// TIA Portal V20 export
VAR_GLOBAL   // PLC tag table "EVT_Const_Gen"
END_VAR
VAR_GLOBAL CONSTANT   // user constants
   EVT_CAPACITY : Int := 1000;   // EVTLOG entries / EVTLOG 항목 수
   EVT_LAST : Int := 999;   // EVTLOG.Entry upper bound / EVTLOG.Entry 상한
   EVT_MIN_LEVEL_DEFAULT : USInt := 2;   // Default Cfg.MinLevel / Cfg.MinLevel 기본값
   EVT_MAX_PER_SCAN_DEFAULT : Int := 32;   // Default Cfg.MaxPerScan / Cfg.MaxPerScan 기본값
   EVT_CATMASK_ALL : DWord := 16#0003FFFE;   // Cfg.CatMask, every category / Cfg.CatMask 전 분류
   EVT_LVL_TRACE : USInt := 0;   // Level TRACE / 레벨 TRACE
   EVT_LVL_DEBUG : USInt := 1;   // Level DEBUG / 레벨 DEBUG
   EVT_LVL_INFO : USInt := 2;   // Level INFO / 레벨 INFO
   EVT_LVL_WARN : USInt := 3;   // Level WARN / 레벨 WARN
   EVT_LVL_ERROR : USInt := 4;   // Level ERROR / 레벨 ERROR
   EVT_CAT_SYS : USInt := 1;   // Category SYS (CatMask bit 1) / 분류 SYS
   EVT_CAT_MODE : USInt := 2;   // Category MODE (CatMask bit 2) / 분류 MODE
   EVT_CAT_STEP : USInt := 3;   // Category STEP (CatMask bit 3) / 분류 STEP
   EVT_CAT_TASK : USInt := 4;   // Category TASK (CatMask bit 4) / 분류 TASK
   EVT_CAT_CMD : USInt := 5;   // Category CMD (CatMask bit 5) / 분류 CMD
   EVT_CAT_ALARM : USInt := 6;   // Category ALARM (CatMask bit 6) / 분류 ALARM
   EVT_CAT_GRIP : USInt := 7;   // Category GRIP (CatMask bit 7) / 분류 GRIP
   EVT_CAT_DRIVE : USInt := 8;   // Category DRIVE (CatMask bit 8) / 분류 DRIVE
   EVT_CAT_SAFETY : USInt := 9;   // Category SAFETY (CatMask bit 9) / 분류 SAFETY
   EVT_CAT_SENSOR : USInt := 10;   // Category SENSOR (CatMask bit 10) / 분류 SENSOR
   EVT_CAT_MEAS : USInt := 11;   // Category MEAS (CatMask bit 11) / 분류 MEAS
   EVT_CAT_ILOCK : USInt := 12;   // Category ILOCK (CatMask bit 12) / 분류 ILOCK
   EVT_CAT_ANTICOL : USInt := 13;   // Category ANTICOL (CatMask bit 13) / 분류 ANTICOL
   EVT_CAT_COMM : USInt := 14;   // Category COMM (CatMask bit 14) / 분류 COMM
   EVT_CAT_DATA : USInt := 15;   // Category DATA (CatMask bit 15) / 분류 DATA
   EVT_CAT_STATION : USInt := 16;   // Category STATION (CatMask bit 16) / 분류 STATION
   EVT_CAT_SCEN : USInt := 17;   // Category SCEN (CatMask bit 17) / 분류 SCEN
   EVT_SYS_STARTUP : UInt := 101;   // SYS INFO / PLC 기동 {a:bits:startup}
   EVT_SYS_PROG_ERROR : UInt := 102;   // SYS ERROR / Programming error : block {src}, Fault_ID {a:hex}, DB {b}
   EVT_SYS_CYCLE_OVERRUN : UInt := 103;   // SYS ERROR / Cycle time error : Fault_ID {a:hex}
   EVT_SYS_CLOCK_SET : UInt := 104;   // SYS WARN / 시계 보정 {a} ms
   EVT_SYS_LOGGER_DROP : UInt := 105;   // SYS WARN / 로거 누락 : Dropped {a} (MaxPerScan 초과)
   EVT_SYS_LOGGER_SLOW : UInt := 106;   // SYS WARN / 로거 실행 시간 MaxRunUs {a} µs
   EVT_MODE_CHANGED : UInt := 201;   // MODE INFO / {b:mode} → {a:mode}
   EVT_MODE_REJECTED : UInt := 202;   // MODE WARN / 모드 요청 거부 {b:mode} → {a:mode}
   EVT_MODE_AUTO_STOP : UInt := 203;   // MODE INFO / AUTO 정지 : {a:auto_stop}
   EVT_MODE_AUTO_START : UInt := 204;   // MODE INFO / AUTO 시작 : {a:start_src}
   EVT_MODE_AUTO_REFUSED : UInt := 205;   // MODE WARN / AUTO 시작 불가 : {a:bits:start_block}
   EVT_MODE_FAULT_RESET : UInt := 206;   // MODE INFO / Fault reset {a:reset_result} (FaultCode[0] {b})
   EVT_MODE_OPTION : UInt := 207;   // MODE WARN / Option {src:option} {a:onoff}
   EVT_MODE_TEACH_BUFF_CLEARED : UInt := 208;   // MODE WARN / Teach 진입 : TASK.Buff {a} 건 삭제
   EVT_MODE_GCS_ONLINE : UInt := 209;   // MODE INFO / GCS_Online {a:onoff}
   EVT_MODE_GRM_PANEL : UInt := 210;   // MODE INFO / GRM {src:grm_panel} {a:onoff}
   EVT_MODE_STATUS_BIT : UInt := 211;   // MODE DEBUG / Status.{src:machine_status} {a:onoff}
   EVT_TASK_ACCEPTED : UInt := 401;   // TASK INFO / 수락 {src:task_type} · Cell {a} · WorkId {b}
   EVT_TASK_REJECTED : UInt := 402;   // TASK WARN / 거부 {src:task_type} : {a:bits:reject} ({b:validation})
   EVT_TASK_HEADER_TIMEOUT : UInt := 403;   // TASK ERROR / 명령 헤더 빈 필드 15 s (F{a})
   EVT_TASK_LOADED : UInt := 404;   // TASK INFO / 시작 {src:task_type} · Cell {a} · WorkId {b}
   EVT_TASK_WAIT_DEADLOCK : UInt := 405;   // TASK WARN / 적재 대기 : 상대 로봇 교착·회피 {a} ms
   EVT_TASK_RESUMED : UInt := 406;   // TASK INFO / 정지 후 재개 → step {a}
   EVT_TASK_CROSSCHECK_FAIL : UInt := 407;   // TASK ERROR / 아이템 교차 확인 실패 F{a}
   EVT_TASK_COMPLETED : UInt := 408;   // TASK INFO / 완료 {src:task_type} · Cell {a} · WorkId {b}
   EVT_TASK_MANUAL_COMPLETE : UInt := 409;   // TASK INFO / 수동 완료 ({src:cmd_src}) : {a:manual_complete} · WorkId {b}
   EVT_TASK_PENDING_END : UInt := 410;   // TASK INFO / CompletePending 해소 : {a:pending_end} · WorkId {b}
   EVT_TASK_CANCELED : UInt := 411;   // TASK INFO / 취소 ({src:cmd_src}) : {a:cancel_result} · WorkId {b}
   EVT_TASK_CANCEL_IGNORED : UInt := 412;   // TASK WARN / AUTO 중 OPC 취소 무시 · WorkId {b}
   EVT_TASK_RESTART_LAST : UInt := 413;   // TASK INFO / 마지막 작업 재시작 · WorkId {b}
   EVT_TASK_TEACH_OVERRIDE : UInt := 414;   // TASK WARN / TeachOverride : {src:override_kind} {a} 위치 갱신
   EVT_TASK_ITEM_CHANGED : UInt := 415;   // TASK INFO / 잡은 아이템 {b} → {a}
   EVT_TASK_CYCLE : UInt := 416;   // TASK INFO / 사이클 ProcessTime {a} ms · Travel {b} mm (flags {src:hex})
   EVT_TASK_STEP_TIMEOUT : UInt := 417;   // TASK WARN / Step {src:task_step} 타임아웃 : WaitCause {a} ({b} ms)
   EVT_TASK_STATUS_BIT : UInt := 418;   // TASK DEBUG / TASK.Status bit {src} {a:onoff}
   EVT_CMD_ALLSTOP : UInt := 501;   // CMD WARN / AllStop {b:onoff} : {a:bits:stop_src}
   EVT_CMD_EMS : UInt := 502;   // CMD ERROR / AllStop_Fast (EMS) {a:onoff}
   EVT_CMD_RESET : UInt := 503;   // CMD INFO / Reset : {a:bits:stop_src}
   EVT_CMD_GCS_START : UInt := 504;   // CMD INFO / GCS Common.Start
   EVT_CMD_BUZZER_STOP : UInt := 505;   // CMD INFO / BuzzerStop
   EVT_CMD_GRIP_LEARN : UInt := 506;   // CMD INFO / Gripper LearnCmd
   EVT_CMD_UNUSED : UInt := 507;   // CMD WARN / 받았지만 처리하지 않는 명령 : {src:unused_cmd}
   EVT_CMD_RESPONSE : UInt := 508;   // CMD INFO / 응답 {b:task_type} SEQ {a}
   EVT_CMD_HMI_TASK_BUTTON : UInt := 509;   // CMD INFO / HMI {src:hmi_task_button}
   EVT_CMD_FUNCTION : UInt := 510;   // CMD INFO / Function {src:function} {a:onoff}
   EVT_CMD_DRIVE_POWER : UInt := 511;   // CMD INFO / {src:axis} PowerOn {a:onoff} (manual)
   EVT_CMD_MANUAL_START : UInt := 512;   // CMD INFO / Manual {src:manual_start} 시작
   EVT_CMD_JOG : UInt := 513;   // CMD DEBUG / {src:axis} Jog {a:hex}
   EVT_ALM_RAISED : UInt := 601;   // ALARM ERROR / {alarm} 발생 (step {b})
   EVT_ALM_CLEARED : UInt := 602;   // ALARM INFO / {alarm} 해제
   EVT_ALM_RESET : UInt := 603;   // ALARM INFO / {src:alarm_area} reset ({a} bits set)
   EVT_ALM_TO_FAULT : UInt := 604;   // ALARM ERROR / FAULT 전환 : 첫 코드 {a}
   EVT_GRIP_REQ : UInt := 701;   // GRIP INFO / 요청 {src:grip_mode} Target {a/10} mm ({b:grip_owner})
   EVT_GRIP_REJECT : UInt := 702;   // GRIP WARN / 요청 거부 {a:grip_err} ({src:grip_owner})
   EVT_GRIP_ABORT : UInt := 703;   // GRIP WARN / 요청 중단 ({src:grip_owner})
   EVT_GRIP_ERROR : UInt := 704;   // GRIP WARN / 실패 {src:grip_err} StopPos {a/10} mm · {b} %
   EVT_GRIP_STATUS : UInt := 705;   // GRIP WARN / {src:grip_status} {a}
   EVT_GRIP_RETRY : UInt := 706;   // GRIP INFO / 재파지 {a} → step {b}
   EVT_GRIP_LEARN : UInt := 707;   // GRIP INFO / Learn {src:learn_phase} LearnError {a} @ {b/10} mm
   EVT_GRIP_THERMAL : UInt := 708;   // GRIP WARN / Thermal {a:onoff}
   EVT_GRIP_STATE : UInt := 709;   // GRIP DEBUG / {b:grip_state} → {a:grip_state}
   EVT_GRIP_ITEM_DETECT : UInt := 710;   // GRIP DEBUG / ItemDetect {a:onoff}
   EVT_GRIP_STEP : UInt := 711;   // GRIP DEBUG / GRIP.Step {b} → {a}
   EVT_GRIP_READY : UInt := 712;   // GRIP WARN / Sense.Ready {a:onoff}
   EVT_DRV_FAULT : UInt := 801;   // DRIVE ERROR / {src:axis} Fault MainCode {a} SubCode {b}
   EVT_DRV_WARNING : UInt := 802;   // DRIVE WARN / {src:axis} Warning MainCode {a} SubCode {b}
   EVT_DRV_FAULT_CLEARED : UInt := 803;   // DRIVE INFO / {src:axis} Fault/Warning 해제
   EVT_DRV_REF_LOST : UInt := 804;   // DRIVE ERROR / {src:axis} Referenced 상실
   EVT_DRV_OVERHEAT : UInt := 805;   // DRIVE WARN / {src:axis} Overheat {a:bits:overheat}
   EVT_DRV_SYNC : UInt := 806;   // DRIVE WARN / X1/X2 sync F{a} (SyncDiff {b/10} mm)
   EVT_DRV_LAG : UInt := 807;   // DRIVE WARN / X lag {a/10} mm ({b:alarm_area})
   EVT_DRV_ENABLE_FAIL : UInt := 808;   // DRIVE ERROR / {src:axis} Enable / encoder F{a}
   EVT_DRV_LIMIT : UInt := 809;   // DRIVE WARN / {src:axis} limit {a:bits:limit}
   EVT_DRV_MDR : UInt := 810;   // DRIVE WARN / MDR {a:bits:mdr}
   EVT_DRV_STATE : UInt := 811;   // DRIVE DEBUG / {src:axis} {a:bits:drive_state}
   EVT_DRV_HOMING_DONE : UInt := 812;   // DRIVE INFO / {src:axis} homing 완료
   EVT_DRV_TARGET_RANGE : UInt := 813;   // DRIVE ERROR / {src:axis} 목표 범위 밖 F{a} (target {b/10} mm)
   EVT_SAFE_EMS : UInt := 901;   // SAFETY ERROR / EMS {a:onoff}
   EVT_SAFE_INPUT : UInt := 902;   // SAFETY WARN / {src:safety_input} {a:onoff}
   EVT_SAFE_IO_FORCE : UInt := 903;   // SAFETY WARN / {src:io_force} {a:onoff}
   EVT_SAFE_OUTPUT : UInt := 904;   // SAFETY DEBUG / Output {src:output} {a:onoff}
   EVT_SNS_MODULE : UInt := 1001;   // SENSOR WARN / Module {src:module} {a:onoff}
   EVT_SNS_BELT : UInt := 1002;   // SENSOR WARN / Belt {src:belt} {a:onoff}
   EVT_SNS_IOLINK_DROP : UInt := 1003;   // SENSOR WARN / IO-Link input {src} 끊김 (누적 {a})
   EVT_SNS_MODULE_DIAG : UInt := 1004;   // SENSOR WARN / Module diag {src:module_diag} : {a:bits:diag_bits}
   EVT_SNS_PDI : UInt := 1005;   // SENSOR DEBUG / {src:pdi} status {a:hex}
   EVT_MEAS_RECORD : UInt := 1101;   // MEAS INFO / 측정 기록 {src:meas_kind} Seq {a} Status {b}
   EVT_MEAS_LOG_RESET : UInt := 1102;   // MEAS WARN / {src:meas_log} reset
   EVT_MEAS_SENSOR : UInt := 1103;   // MEAS WARN / Laser {src} : {a:bits:laser_flag}
   EVT_MEAS_SLOWDOWN : UInt := 1104;   // MEAS DEBUG / ZSlowDown {src:slowdown}
   EVT_ILK_TARGET : UInt := 1201;   // ILOCK INFO / WorkCell {a} · WorkType {b:hex}
   EVT_ILK_PI : UInt := 1202;   // ILOCK INFO / PI {a:bits:pi_bits} (이전 {b:bits:pi_bits})
   EVT_ILK_PO : UInt := 1203;   // ILOCK INFO / PO {a:bits:po_bits} (이전 {b:bits:po_bits})
   EVT_ILK_TIMEOUT : UInt := 1204;   // ILOCK ERROR / Interlock timeout F{a} (step {src})
   EVT_ACL_TARGET_SHIFT : UInt := 1301;   // ANTICOL INFO / 회피 목표 변경 X {a/10} → {b/10} mm
   EVT_ACL_APPROACH : UInt := 1302;   // ANTICOL WARN / 상대 로봇 접근·교착 F{a}
   EVT_ACL_LIMIT : UInt := 1303;   // ANTICOL ERROR / 충돌 한계 F{a}
   EVT_ACL_SPEED : UInt := 1304;   // ANTICOL INFO / SpeedFactor {src:speed_kind} {b} → {a} %
   EVT_ACL_AVOID : UInt := 1305;   // ANTICOL DEBUG / AvoidReq {a:onoff}
   EVT_COM_LINK : UInt := 1401;   // COMM WARN / {src:peer} link {a:onoff} (끊김 {b} ms)
   EVT_COM_BLOCK_ERR : UInt := 1402;   // COMM WARN / {src:comm_block} error STATUS {a:hex}
   EVT_COM_CMD_FRAME : UInt := 1403;   // COMM INFO / GRM 명령 프레임 수신 {b:task_type}
   EVT_COM_HEARTBEAT : UInt := 1404;   // COMM WARN / {src:peer} heartbeat {b:stall} ({a} ms)
   EVT_COM_XY_STOP : UInt := 1405;   // COMM WARN / 통신 끊김으로 XY 정지 (W{a})
   EVT_COM_SOCK : UInt := 1406;   // COMM INFO / Socket slot {src} {a:sock_state} (LastErr {b})
   EVT_COM_GET_FAIL : UInt := 1407;   // COMM DEBUG / GET NDR 없음 STATUS {a:hex}
   EVT_DATA_CSV : UInt := 1501;   // DATA INFO / CSV {src:csv_kind} : {a:csv_result} (STATUS {b:hex})
   EVT_DATA_PARA_HMI : UInt := 1502;   // DATA INFO / HMI p{src} {b/100} → {a/100}
   EVT_DATA_PARA_HOMING : UInt := 1503;   // DATA WARN / Homing 이 {src:para} 를 씀 {b/100} → {a/100}
   EVT_DATA_PARA_ADJUST : UInt := 1504;   // DATA WARN / Adjust 가 {src:para} 를 씀 {b/100} → {a/100}
   EVT_DATA_PARA_ZCAL : UInt := 1505;   // DATA WARN / Laser ZCal 이 {src:para} 를 씀 {b/100} → {a/100}
   EVT_DATA_PARA_AUTOCAL : UInt := 1506;   // DATA WARN / Laser AutoCal 이 {src:para} 를 씀 {b/100} → {a/100}
   EVT_DATA_PARA_CALZ : UInt := 1507;   // DATA WARN / CalibrationZ 가 {src:para} 를 씀 {b/100} → {a/100}
   EVT_DATA_PARA_SECTION : UInt := 1508;   // DATA INFO / PARA.{src:para_section} 변경 (checksum {b:hex} → {a:hex})
   EVT_DATA_PARA_SPEED : UInt := 1509;   // DATA INFO / HMI SpeedSet {src:axis} index {a} 변경
   EVT_ALARM_AREA_FAULT : UInt := 1;   // alarm_area = FAULT
   EVT_ALARM_AREA_WARN : UInt := 2;   // alarm_area = WARN
   EVT_ALARM_AREA_EVENT : UInt := 3;   // alarm_area = EVENT
   EVT_ALARM_AREA_TASK : UInt := 4;   // alarm_area = TASK
   EVT_AUTO_STOP_PB_STOP : UInt := 1;   // auto_stop = PB_Stop
   EVT_AUTO_STOP_ALLSTOP : UInt := 2;   // auto_stop = AllStop
   EVT_AUTO_STOP_EMS : UInt := 3;   // auto_stop = EMS
   EVT_AUTO_STOP_SSW_AUTO_OFF : UInt := 4;   // auto_stop = SSW_Auto off
   EVT_CANCEL_RESULT_OK : UInt := 1;   // cancel_result = OK
   EVT_CANCEL_RESULT_REFUSED_F6020 : UInt := 2;   // cancel_result = Refused (F6020)
   EVT_CMD_SRC_OPC : UInt := 1;   // cmd_src = OPC
   EVT_CMD_SRC_HMI : UInt := 2;   // cmd_src = HMI
   EVT_CMD_SRC_HMI_FORCE : UInt := 3;   // cmd_src = HMI Force
   EVT_CMD_SRC_SOCKET : UInt := 4;   // cmd_src = Socket
   EVT_CSV_RESULT_IMPORT_REQUEST : UInt := 1;   // csv_result = Import request
   EVT_CSV_RESULT_IMPORT_DONE : UInt := 2;   // csv_result = Import done
   EVT_CSV_RESULT_IMPORT_TIMEOUT : UInt := 3;   // csv_result = Import timeout
   EVT_CSV_RESULT_FILE_MISSING_DEFAULTS : UInt := 4;   // csv_result = File missing -> defaults
   EVT_CSV_RESULT_IMPORT_ERROR_TREATED_AS_DONE : UInt := 5;   // csv_result = Import error (treated as done)
   EVT_CSV_RESULT_EXPORT : UInt := 6;   // csv_result = Export
   EVT_CSV_RESULT_EXPORT_ERROR : UInt := 7;   // csv_result = Export error
   EVT_LEARN_PHASE_ACCEPTED : UInt := 1;   // learn_phase = Accepted
   EVT_LEARN_PHASE_DONE : UInt := 2;   // learn_phase = Done
   EVT_LEARN_PHASE_ERROR : UInt := 3;   // learn_phase = Error
   EVT_MANUAL_COMPLETE_REQUESTED : UInt := 1;   // manual_complete = Requested
   EVT_MANUAL_COMPLETE_REFUSED_AUTO_W6026 : UInt := 2;   // manual_complete = Refused AUTO (W6026)
   EVT_MANUAL_COMPLETE_GRIP_NG_F6022 : UInt := 3;   // manual_complete = Grip NG (F6022)
   EVT_MANUAL_COMPLETE_NO_ITEM_F6018 : UInt := 4;   // manual_complete = No item (F6018)
   EVT_MANUAL_COMPLETE_PENDING_CV_HANDOVER : UInt := 5;   // manual_complete = Pending CV handover
   EVT_MANUAL_COMPLETE_DONE : UInt := 6;   // manual_complete = Done
   EVT_PARA_SENSOR_GIDL_ZOFFSET : UInt := 1;   // para = Sensor.GIDL_ZOffset
   EVT_PARA_SENSOR_GIDF_ZOFFSET : UInt := 2;   // para = Sensor.GIDF_ZOffset
   EVT_PARA_SENSOR_GIDR_ZOFFSET : UInt := 3;   // para = Sensor.GIDR_ZOffset
   EVT_PARA_SENSOR_GIDB_ZOFFSET : UInt := 4;   // para = Sensor.GIDB_ZOffset
   EVT_PARA_DRIVE_HOMEPOS_X : UInt := 11;   // para = Drive.HomePos[X]
   EVT_PARA_DRIVE_HOMEPOS_Y : UInt := 12;   // para = Drive.HomePos[Y]
   EVT_PARA_DRIVE_HOMEPOS_Z : UInt := 13;   // para = Drive.HomePos[Z]
   EVT_PARA_DRIVE_HOMEPOS_G : UInt := 14;   // para = Drive.HomePos[G]
   EVT_PARA_DRIVE_RANGEMIN_X : UInt := 21;   // para = Drive.RangeMin[X]
   EVT_PARA_DRIVE_RANGEMIN_Y : UInt := 22;   // para = Drive.RangeMin[Y]
   EVT_PARA_DRIVE_RANGEMIN_Z : UInt := 23;   // para = Drive.RangeMin[Z]
   EVT_PARA_DRIVE_RANGEMIN_G : UInt := 24;   // para = Drive.RangeMin[G]
   EVT_PARA_DRIVE_RANGEMAX_X : UInt := 31;   // para = Drive.RangeMax[X]
   EVT_PARA_DRIVE_RANGEMAX_Y : UInt := 32;   // para = Drive.RangeMax[Y]
   EVT_PARA_DRIVE_RANGEMAX_Z : UInt := 33;   // para = Drive.RangeMax[Z]
   EVT_PARA_DRIVE_RANGEMAX_G : UInt := 34;   // para = Drive.RangeMax[G]
   EVT_PARA_DRIVE_MCS_TO_ACS_Z_0 : UInt := 41;   // para = Drive.MCS_TO_ACS[Z,0]
   EVT_PARA_DRIVE_MCS_TO_ACS_Z_1 : UInt := 42;   // para = Drive.MCS_TO_ACS[Z,1]
   EVT_PARA_DRIVE_MCS_TO_ACS_Z_2 : UInt := 43;   // para = Drive.MCS_TO_ACS[Z,2]
   EVT_PARA_DRIVE_ACS_TO_MCS_Z_0 : UInt := 44;   // para = Drive.ACS_TO_MCS[Z,0]
   EVT_PARA_DRIVE_ACS_TO_MCS_Z_1 : UInt := 45;   // para = Drive.ACS_TO_MCS[Z,1]
   EVT_PARA_DRIVE_ACS_TO_MCS_Z_2 : UInt := 46;   // para = Drive.ACS_TO_MCS[Z,2]
   EVT_PARA_MACHINE_XLENGTHFRONT : UInt := 51;   // para = Machine.XLengthFront
   EVT_PARA_MACHINE_XLENGTHREAR : UInt := 52;   // para = Machine.XLengthRear
   EVT_PARA_SENSOR_XACF_OFFSET : UInt := 53;   // para = Sensor.XACF_Offset
   EVT_PARA_SENSOR_XACR_OFFSET : UInt := 54;   // para = Sensor.XACR_Offset
   EVT_PARA_SENSOR_FLD_OFFSET : UInt := 55;   // para = Sensor.FLD_Offset
   EVT_PARA_MACHINE_G_OFFSET : UInt := 56;   // para = Machine.G_Offset
   EVT_PENDING_END_CV_HANDOVER : UInt := 1;   // pending_end = CV handover
   EVT_PENDING_END_AUTO_FORCED_W6024 : UInt := 2;   // pending_end = AUTO forced (W6024)
   EVT_PENDING_END_TIMEOUT_W6024 : UInt := 3;   // pending_end = Timeout (W6024)
   EVT_PENDING_END_DROPPED : UInt := 4;   // pending_end = Dropped
   EVT_PROC_TASK : UInt := 20;   // proc = Task
   EVT_PROC_INIT : UInt := 100;   // proc = Init
   EVT_PROC_CHANGEIP : UInt := 110;   // proc = ChangeIP
   EVT_PROC_HOMINGX : UInt := 121;   // proc = HomingX
   EVT_PROC_HOMINGY : UInt := 122;   // proc = HomingY
   EVT_PROC_HOMINGZ : UInt := 123;   // proc = HomingZ
   EVT_PROC_HOMINGG : UInt := 124;   // proc = HomingG
   EVT_PROC_INITPOS : UInt := 130;   // proc = InitPos
   EVT_PROC_MEASUREITEM : UInt := 140;   // proc = MeasureItem
   EVT_PROC_MANUALMEASURE : UInt := 141;   // proc = ManualMeasure
   EVT_PROC_CALIBRATIONZ : UInt := 150;   // proc = CalibrationZ
   EVT_PROC_CELLORIGINX : UInt := 161;   // proc = CellOriginX
   EVT_PROC_CELLORIGINY : UInt := 162;   // proc = CellOriginY
   EVT_RESET_RESULT_TRY : UInt := 1;   // reset_result = Try
   EVT_RESET_RESULT_OK : UInt := 2;   // reset_result = OK
   EVT_RESET_RESULT_FAIL : UInt := 3;   // reset_result = Fail
   EVT_START_BLOCK_ROBOTUSE : UInt := 0;   // start_block = RobotUse
   EVT_START_BLOCK_POWERONDRIVE : UInt := 1;   // start_block = PowerOnDrive
   EVT_START_BLOCK_DRIVESYNC : UInt := 2;   // start_block = DriveSync
   EVT_START_BLOCK_GRM_CONNECTED : UInt := 3;   // start_block = GRM_Connected
   EVT_START_SRC_PB_START : UInt := 1;   // start_src = PB_Start
   EVT_START_SRC_GCS_COMMON_START : UInt := 2;   // start_src = GCS Common.Start
   EVT_UNUSED_CMD_STOP_FAST : UInt := 1;   // unused_cmd = Stop.Fast
   EVT_UNUSED_CMD_STOP_CYCLE : UInt := 2;   // unused_cmd = Stop.Cycle
   EVT_UNUSED_CMD_COMMON_INITIALIZING : UInt := 3;   // unused_cmd = Common.Initializing
   EVT_UNUSED_CMD_JOG : UInt := 4;   // unused_cmd = Jog
   EVT_UNUSED_CMD_HOME : UInt := 5;   // unused_cmd = Home
   EVT_UNUSED_CMD_MAINTPOS : UInt := 6;   // unused_cmd = MaintPos
   EVT_UNUSED_CMD_CELLORIGIN : UInt := 7;   // unused_cmd = CellOrigin
   EVT_UNUSED_CMD_CHANGEMODE : UInt := 8;   // unused_cmd = ChangeMode
END_VAR
